TYPE ST_MotionDefaults :
	STRUCT
		DefaultResetTask : CoEResetTask				  := (Name := 'MC Reset (CoE)');
		DefaultHomeTask	 : MotionHomeTask_SetZeroHere := (Name := 'MC Home');
		DefaultStopTask	 : StopTask					  := (Name := 'MC Stop');
	END_STRUCT
END_TYPE

(* stored: Version 1.1.0.1, ProductVersion 3.1.4026.18
   DUT ST_MotionDefaults: Id {c9d96df1-da2a-43a5-8f71-11090870ce3d} *)
